// TIA Portal V20 export
TYPE "HMIAxisCtrl_typeOutputs"
TITLE = HMIAxisCtrl_typeOutputs
// Support: tech.team.motioncontrol@siemens.com 
// Fax: +49 (0) 9131/98-1297
   STRUCT
      valid : Bool;   // TRUE: Valid set of outputs available at the FB
      busy : Bool;   // TRUE: FB is working and new output values can be expected
      error : Bool;   // TRUE: An error occurred while processing the FB
      status : Word;   // Current status of FB
      axisEnabled : Bool;   // TRUE: The technology object is enabled. Motion commands can be executed.
      resetActive : Bool;   // TRUE: Reset/Restart of the axis is active
      commandBusy : Bool;   // TRUE: The selected basic motion command is being executed
      commandDone : Bool;   // TRUE: The selected basic motion command has completed without error
      commandAborted : Bool;   // TRUE: The selected basic motion command has been aborted
      inVelocity : Bool;   // TRUE: The setpoint velocity/speed was reached and will be maintained
      inLimitation : Bool;   // TRUE: The drive is operating at the force/torque limit
      homingCommandBusy : Bool;   // TRUE: Homing command is being executed
      homingCommandDone : Bool;   // TRUE: Homing command has completed without error
      homingCommandAborted : Bool;   // TRUE: Homing command has been aborted
      superimposedBusy : Bool;   // TRUE: The selected superimposed motion command is being executed
      superimposedDone : Bool;   // TRUE: The selected superimposed motion command has completed without error
      superimposedAborted : Bool;   // TRUE: The selected superimposed motion command has been aborted
      inClamping : Bool;   // TRUE: The drive is kept at the fixed stop (clamping), the axis position is within the positioning tolerance
      startSync : Bool;   // TRUE: The axis is synchronizing to the leading axis
      inSync : Bool;   // TRUE: The axis is synchronized to the leading axis
      inSimulation : Bool;   // TRUE: Synchronous operation is being simulated
      jogSelected : Bool;   // TRUE: Jogging is active
      moveVelocitySelected : Bool;   // TRUE: Moving with constant velocity/speed is active
      stopSelected : Bool;   // TRUE: Stopping is active
      fastStopSelected : Bool;   // TRUE: Stopping is active (with fastStop dynamics)
      torqueLimitingSelected : Bool;   // TRUE: Force/Torque limiting is active
      homingSelected : Bool;   // TRUE: Homing is active
      posRelativeSelected : Bool;   // TRUE: Relative positioning is active
      posAbsoluteSelected : Bool;   // TRUE: Absolute positioning is active
      posSuperimposedSelected : Bool;   // TRUE: Superimposed positioning is active
      gearInRelativeSelected : Bool;   // TRUE: Relative gearing is active
      gearInAbsoluteSelected : Bool;   // TRUE: Absolute gearing is active
      camInSelected : Bool;   // TRUE: Camming is active
      phasingSelected : Bool;   // TRUE: Phasing is active
   END_STRUCT;
END_TYPE
